{attribute 'GeneratedUsingTerminal: EM7004-0000-0017'}
{attribute addProperty BoxType "EM7004-0000-0017"}
{attribute addProperty Id "PLS_EnabledBOOL1Unequal_SI_0BOOL1"}
{attribute addProperty CRC "2284459279"}
{attribute addProperty Size "2"}
TYPE Status_882A150F :
STRUCT
	{attribute addProperty Name "PLS_Enabled"}
	PLS_Enabled : BOOL;
	{attribute addProperty Name "Unequal_SI_0"}
	Unequal_SI_0 : BOOL;
END_STRUCT
END_TYPE
